// Mitsubishi GX Works2 project: 20150618   PLC: Q03UDV

PROGRAM P1
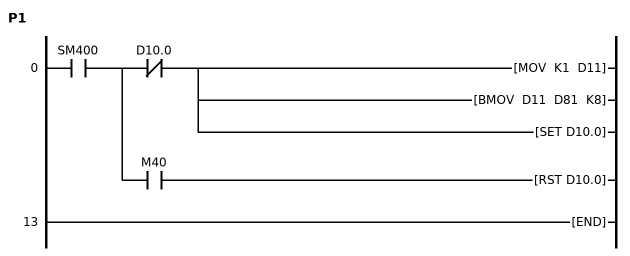
0     LD      SM400
      MPS
      ANI     D10.0
      MOV     K1 D11
      BMOV    D11 D81 K8
      SET     D10.0
      MPP
      AND     M40
      RST     D10.0
13    END
END_PROGRAM

PROGRAM P2
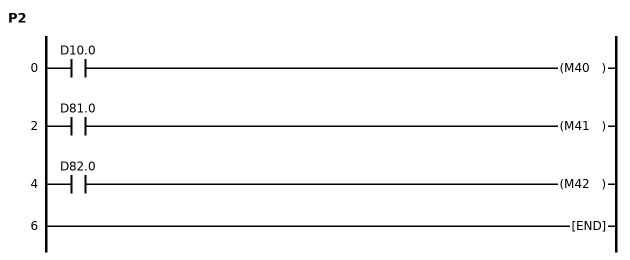
0     LD      D10.0
      OUT     M40
2     LD      D81.0
      OUT     M41
4     LD      D82.0
      OUT     M42
6     END
END_PROGRAM
